// TwinCAT 3 PLC project Untitled1
// ProgramVersion: 3.1.4023.0
// libraries:
//   Tc2_EthernetIP, * (Beckhoff Automation GmbH)
//   Tc2_Standard, * (Beckhoff Automation GmbH)
//   Tc2_System, * (Beckhoff Automation GmbH)
//   Tc3_Module, * (Beckhoff Automation GmbH)
// project tree:
//   GVLs/ GVL.TcGVL
//   / PlcTask.TcTTO
//   POUs/ MAIN.TcPOU

CONFIGURATION Untitled1
    RESOURCE PLC ON TwinCAT3
        TASK PlcTask(INTERVAL := T#10ms, PRIORITY := 20);
        PROGRAM MAIN WITH PlcTask : MAIN;
    END_RESOURCE
END_CONFIGURATION

// ---- GVLs/GVL.TcGVL
{attribute 'qualified_only'}
VAR_GLOBAL
	Input_State AT %I*: UINT;
	Output_State AT %Q*: UINT;
	ConnState AT %I*: UDINT;
	ConnCtrl AT %Q*: UDINT;
	Input_100 AT %I*: ARRAY[0..100] OF BYTE;
	Output_100 AT %Q*: ARRAY[0..100] OF BYTE;
END_VAR

// ---- POUs/MAIN.TcPOU
PROGRAM MAIN
VAR
	sad: DINT;
END_VAR

sad := 1 +sad;

END_PROGRAM
